{attribute 'GeneratedUsingTerminal: EJ6910-0000-0018'}
{attribute addProperty BoxType "EJ6910-0000-0018"}
{attribute addProperty Id "FSLOGIC_InputsAT %I*FSLOGIC_Inputs_EEE9388E2FSLOGIC_OutputsAT %I*EMPTY_STRUCTURE0WcStateAT %I*WcState_9091E0EB2InfoDataAT %I*InfoData_94A18F5E2"}
{attribute addProperty CRC "1258662764"}
{attribute addProperty Size "6"}
TYPE EJ6910_4B05AB6C EXTENDS EtcSlaveTerminalBase_947E5A46 :
STRUCT
	{attribute addProperty Name "FSLOGIC_Inputs"}
	FSLOGIC_Inputs : FSLOGIC_Inputs_EEE9388E;
	{attribute addProperty Name "FSLOGIC_Outputs"}
	FSLOGIC_Outputs : EMPTY_STRUCTURE;
	{attribute addProperty Name "WcState"}
	WcState : WcState_9091E0EB;
	{attribute addProperty Name "InfoData"}
	InfoData : InfoData_94A18F5E;
END_STRUCT
END_TYPE

(* stored: Version 1.2.0.0, ProductVersion 3.1.4024.9
   DUT EJ6910_4B05AB6C: Id {4826695d-0b46-407b-8435-b76419c800b6} *)
